Yaskawa INFORM job: GAUSSIANMOVING2.JBI

/JOB
//NAME GAUSSIANMOVING2
//POS
///NPOS 0,0,0,121,0,0
///TOOL 0
///POSTYPE ROBOT
///RECTAN
///RCONF 0,0,0,0,0,0,0,0,0,0,0,0,0,0,0,0,0,0,0,0,0,0,0,0
P00000=10.000,0.000,0.000,0.0000,0.0000,0.0000
///POSTYPE BASE
///TOOL0
P00001=0652.35187878,0006.95945011,0523.09500000,0000.00000000,0000.00400000,0180.00000000,
P00002=0652.29694326,0006.95464388,0523.09500000,0000.00000000,0000.00400000,0180.00000000,
P00003=0652.22427337,0006.94828609,0523.09500000,0000.00000000,0000.00400000,0180.00000000,
P00004=0652.12909978,0006.93995948,0523.09500000,0000.00000000,0000.00400000,0180.00000000,
P00005=0652.00569299,0006.92916278,0523.09500000,0000.00000000,0000.00400000,0180.00000000,
P00006=0651.84726850,0006.91530243,0523.09500000,0000.00000000,0000.00400000,0180.00000000,
P00007=0651.64591172,0006.89768600,0523.09500000,0000.00000000,0000.00400000,0180.00000000,
P00008=0651.39253259,0006.87551820,0523.09500000,0000.00000000,0000.00400000,0180.00000000,
P00009=0651.07686056,0006.84790047,0523.09500000,0000.00000000,0000.00400000,0180.00000000,
P00010=0650.68749098,0006.81383505,0523.09500000,0000.00000000,0000.00400000,0180.00000000,
P00011=0650.21199308,0006.77223437,0523.09500000,0000.00000000,0000.00400000,0180.00000000,
P00012=0649.63708838,0006.72193673,0523.09500000,0000.00000000,0000.00400000,0180.00000000,
P00013=0648.94890563,0006.66172854,0523.09500000,0000.00000000,0000.00400000,0180.00000000,
P00014=0648.13331474,0006.59037358,0523.09500000,0000.00000000,0000.00400000,0180.00000000,
P00015=0647.17633747,0006.50664892,0523.09500000,0000.00000000,0000.00400000,0180.00000000,
P00016=0646.06462739,0006.40938689,0523.09500000,0000.00000000,0000.00400000,0180.00000000,
P00017=0644.78600549,0006.29752197,0523.09500000,0000.00000000,0000.00400000,0180.00000000,
P00018=0643.33003222,0006.17014081,0523.09500000,0000.00000000,0000.00400000,0180.00000000,
P00019=0641.68859100,0006.02653332,0523.09500000,0000.00000000,0000.00400000,0180.00000000,
P00020=0639.85645402,0005.86624210,0523.09500000,0000.00000000,0000.00400000,0180.00000000,
P00021=0637.83179817,0005.68910767,0523.09500000,0000.00000000,0000.00400000,0180.00000000,
P00022=0635.61663786,0005.49530625,0523.09500000,0000.00000000,0000.00400000,0180.00000000,
P00023=0633.21714325,0005.28537767,0523.09500000,0000.00000000,0000.00400000,0180.00000000,
P00024=0630.64381570,0005.06024069,0523.09500000,0000.00000000,0000.00400000,0180.00000000,
P00025=0627.91149903,0004.82119395,0523.09500000,0000.00000000,0000.00400000,0180.00000000,
P00026=0625.03921312,0004.56990150,0523.09500000,0000.00000000,0000.00400000,0180.00000000,
P00027=0622.04980661,0004.30836232,0523.09500000,0000.00000000,0000.00400000,0180.00000000,
P00028=0618.96943611,0004.03886482,0523.09500000,0000.00000000,0000.00400000,0180.00000000,
P00029=0615.82689035,0003.76392769,0523.09500000,0000.00000000,0000.00400000,0180.00000000,
P00030=0612.65278792,0003.48622971,0523.09500000,0000.00000000,0000.00400000,0180.00000000,
P00031=0609.47868550,0003.20853173,0523.09500000,0000.00000000,0000.00400000,0180.00000000,
P00032=0606.33613974,0002.93359460,0523.09500000,0000.00000000,0000.00400000,0180.00000000,
P00033=0603.25576923,0002.66409710,0523.09500000,0000.00000000,0000.00400000,0180.00000000,
P00034=0600.26636273,0002.40255792,0523.09500000,0000.00000000,0000.00400000,0180.00000000,
P00035=0597.39407682,0002.15126547,0523.09500000,0000.00000000,0000.00400000,0180.00000000,
P00036=0594.66176015,0001.91221873,0523.09500000,0000.00000000,0000.00400000,0180.00000000,
P00037=0592.08843260,0001.68708175,0523.09500000,0000.00000000,0000.00400000,0180.00000000,
P00038=0589.68893799,0001.47715317,0523.09500000,0000.00000000,0000.00400000,0180.00000000,
P00039=0587.47377768,0001.28335175,0523.09500000,0000.00000000,0000.00400000,0180.00000000,
P00040=0585.44912182,0001.10621732,0523.09500000,0000.00000000,0000.00400000,0180.00000000,
P00041=0583.61698485,0000.94592610,0523.09500000,0000.00000000,0000.00400000,0180.00000000,
P00042=0581.97554363,0000.80231861,0523.09500000,0000.00000000,0000.00400000,0180.00000000,
P00043=0580.51957036,0000.67493745,0523.09500000,0000.00000000,0000.00400000,0180.00000000,
P00044=0579.24094846,0000.56307253,0523.09500000,0000.00000000,0000.00400000,0180.00000000,
P00045=0578.12923838,0000.46581050,0523.09500000,0000.00000000,0000.00400000,0180.00000000,
P00046=0577.17226111,0000.38208584,0523.09500000,0000.00000000,0000.00400000,0180.00000000,
P00047=0576.35667022,0000.31073088,0523.09500000,0000.00000000,0000.00400000,0180.00000000,
P00048=0575.66848747,0000.25052269,0523.09500000,0000.00000000,0000.00400000,0180.00000000,
P00049=0575.09358277,0000.20022505,0523.09500000,0000.00000000,0000.00400000,0180.00000000,
P00050=0574.61808487,0000.15862437,0523.09500000,0000.00000000,0000.00400000,0180.00000000,
P00051=0574.22871528,0000.12455895,0523.09500000,0000.00000000,0000.00400000,0180.00000000,
P00052=0573.91304326,0000.09694122,0523.09500000,0000.00000000,0000.00400000,0180.00000000,
P00053=0573.65966412,0000.07477342,0523.09500000,0000.00000000,0000.00400000,0180.00000000,
P00054=0573.45830735,0000.05715699,0523.09500000,0000.00000000,0000.00400000,0180.00000000,
P00055=0573.29988285,0000.04329664,0523.09500000,0000.00000000,0000.00400000,0180.00000000,
P00056=0573.17647606,0000.03249994,0523.09500000,0000.00000000,0000.00400000,0180.00000000,
P00057=0573.08130247,0000.02417333,0523.09500000,0000.00000000,0000.00400000,0180.00000000,
P00058=0573.00863258,0000.01781554,0523.09500000,0000.00000000,0000.00400000,0180.00000000,
P00059=0572.95369707,0000.01300931,0523.09500000,0000.00000000,0000.00400000,0180.00000000,
P00060=0572.91258090,0000.00941211,0523.09500000,0000.00000000,0000.00400000,0180.00000000,
///TOOL1
P00061=0667.35246409,0026.78692869,0908.48000000,0180.00000000,0000.00000000,0000.00000000
P00062=0667.35742094,0026.76842948,0908.48000000,0180.00000000,0000.00000000,0000.00000000
P00063=0667.36397796,0026.74395834,0908.48000000,0180.00000000,0000.00000000,0000.00000000
P00064=0667.37256550,0026.71190921,0908.48000000,0180.00000000,0000.00000000,0000.00000000
P00065=0667.38370053,0026.67035272,0908.48000000,0180.00000000,0000.00000000,0000.00000000
P00066=0667.39799521,0026.61700424,0908.48000000,0180.00000000,0000.00000000,0000.00000000
P00067=0667.41616369,0026.54919856,0908.48000000,0180.00000000,0000.00000000,0000.00000000
P00068=0667.43902615,0026.46387468,0908.48000000,0180.00000000,0000.00000000,0000.00000000
P00069=0667.46750932,0026.35757404,0908.48000000,0180.00000000,0000.00000000,0000.00000000
P00070=0667.50264224,0026.22645619,0908.48000000,0180.00000000,0000.00000000,0000.00000000
P00071=0667.54554654,0026.06633516,0908.48000000,0180.00000000,0000.00000000,0000.00000000
P00072=0667.59742035,0025.87273949,0908.48000000,0180.00000000,0000.00000000,0000.00000000
P00073=0667.65951526,0025.64099813,0908.48000000,0180.00000000,0000.00000000,0000.00000000
P00074=0667.73310624,0025.36635284,0908.48000000,0180.00000000,0000.00000000,0000.00000000
P00075=0667.81945455,0025.04409656,0908.48000000,0180.00000000,0000.00000000,0000.00000000
P00076=0667.91976445,0024.66973493,0908.48000000,0180.00000000,0000.00000000,0000.00000000
P00077=0668.03513484,0024.23916677,0908.48000000,0180.00000000,0000.00000000,0000.00000000
P00078=0668.16650769,0023.74887660,0908.48000000,0180.00000000,0000.00000000,0000.00000000
P00079=0668.31461537,0023.19613124,0908.48000000,0180.00000000,0000.00000000,0000.00000000
P00080=0668.47992957,0022.57917023,0908.48000000,0180.00000000,0000.00000000,0000.00000000
P00081=0668.66261480,0021.89737966,0908.48000000,0180.00000000,0000.00000000,0000.00000000
P00082=0668.86248931,0021.15143787,0908.48000000,0180.00000000,0000.00000000,0000.00000000
P00083=0669.07899634,0020.34342262,0908.48000000,0180.00000000,0000.00000000,0000.00000000
P00084=0669.31118836,0019.47687018,0908.48000000,0180.00000000,0000.00000000,0000.00000000
P00085=0669.55772602,0018.55677912,0908.48000000,0180.00000000,0000.00000000,0000.00000000
P00086=0669.81689314,0017.58955428,0908.48000000,0180.00000000,0000.00000000,0000.00000000
P00087=0670.08662808,0016.58288978,0908.48000000,0180.00000000,0000.00000000,0000.00000000
P00088=0670.36457072,0015.54559370,0908.48000000,0180.00000000,0000.00000000,0000.00000000
P00089=0670.64812346,0014.48736049,0908.48000000,0180.00000000,0000.00000000,0000.00000000
P00090=0670.93452356,0013.41850076,0908.48000000,0180.00000000,0000.00000000,0000.00000000
P00091=0671.22092366,0012.34964103,0908.48000000,0180.00000000,0000.00000000,0000.00000000
P00092=0671.50447639,0011.29140782,0908.48000000,0180.00000000,0000.00000000,0000.00000000
P00093=0671.78241904,0010.25411174,0908.48000000,0180.00000000,0000.00000000,0000.00000000
P00094=0672.05215398,0009.24744724,0908.48000000,0180.00000000,0000.00000000,0000.00000000
P00095=0672.31132110,0008.28022240,0908.48000000,0180.00000000,0000.00000000,0000.00000000
P00096=0672.55785875,0007.36013134,0908.48000000,0180.00000000,0000.00000000,0000.00000000
P00097=0672.79005078,0006.49357890,0908.48000000,0180.00000000,0000.00000000,0000.00000000
P00098=0673.00655781,0005.68556365,0908.48000000,0180.00000000,0000.00000000,0000.00000000
P00099=0673.20643231,0004.93962186,0908.48000000,0180.00000000,0000.00000000,0000.00000000
P00100=0673.38911754,0004.25783129,0908.48000000,0180.00000000,0000.00000000,0000.00000000
P00101=0673.55443175,0003.64087028,0908.48000000,0180.00000000,0000.00000000,0000.00000000
P00102=0673.70253942,0003.08812491,0908.48000000,0180.00000000,0000.00000000,0000.00000000
P00103=0673.83391228,0002.59783475,0908.48000000,0180.00000000,0000.00000000,0000.00000000
P00104=0673.94928267,0002.16726659,0908.48000000,0180.00000000,0000.00000000,0000.00000000
P00105=0674.04959256,0001.79290496,0908.48000000,0180.00000000,0000.00000000,0000.00000000
P00106=0674.13594088,0001.47064867,0908.48000000,0180.00000000,0000.00000000,0000.00000000
P00107=0674.20953186,0001.19600339,0908.48000000,0180.00000000,0000.00000000,0000.00000000
P00108=0674.27162677,0000.96426203,0908.48000000,0180.00000000,0000.00000000,0000.00000000
P00109=0674.32350057,0000.77066636,0908.48000000,0180.00000000,0000.00000000,0000.00000000
P00110=0674.36640487,0000.61054533,0908.48000000,0180.00000000,0000.00000000,0000.00000000
P00111=0674.40153779,0000.47942748,0908.48000000,0180.00000000,0000.00000000,0000.00000000
P00112=0674.43002096,0000.37312684,0908.48000000,0180.00000000,0000.00000000,0000.00000000
P00113=0674.45288343,0000.28780296,0908.48000000,0180.00000000,0000.00000000,0000.00000000
P00114=0674.47105191,0000.21999728,0908.48000000,0180.00000000,0000.00000000,0000.00000000
P00115=0674.48534659,0000.16664880,0908.48000000,0180.00000000,0000.00000000,0000.00000000
P00116=0674.49648162,0000.12509231,0908.48000000,0180.00000000,0000.00000000,0000.00000000
P00117=0674.50506915,0000.09304318,0908.48000000,0180.00000000,0000.00000000,0000.00000000
P00118=0674.51162618,0000.06857204,0908.48000000,0180.00000000,0000.00000000,0000.00000000
P00119=0674.51658302,0000.05007283,0908.48000000,0180.00000000,0000.00000000,0000.00000000
P00120=0674.52029295,0000.03622722,0908.48000000,0180.00000000,0000.00000000,0000.00000000
//INST
///DATE 2017/03/31 08:11
///COMM PLAYINGTWOROBOTS
///ATTR SC,RW
///GROUP1 RB1
///GROUP2 RB2
NOP
DOUT OT#(16) OFF
DOUT OT#(15) ON
DOUT OT#(16) ON
MOVL P00001 V=0003.4465852  +MOVL P00061 V=0001.1969865
MOVL P00002 V=0004.5592174  +MOVL P00062 V=0001.5833996
MOVL P00003 V=0005.9710711  +MOVL P00063 V=0002.0737312
MOVL P00004 V=0007.7423865  +MOVL P00064 V=0002.6889026
MOVL P00005 V=0009.9393530  +MOVL P00065 V=0003.4519011
MOVL P00006 V=0012.6328705  +MOVL P00066 V=0004.3873499
MOVL P00007 V=0015.8966875  +MOVL P00067 V=0005.5208616
MOVL P00008 V=0019.8048652  +MOVL P00068 V=0006.8781575
MOVL P00009 V=0024.4285569  +MOVL P00069 V=0008.4839488
MOVL P00010 V=0029.8321393  +MOVL P00070 V=0010.3605933
MOVL P00011 V=0036.0687965  +MOVL P00071 V=0012.5265616
MOVL P00012 V=0043.1757182  +MOVL P00072 V=0014.9947696
MOVL P00013 V=0051.1691447  +MOVL P00073 V=0017.7708575
MOVL P00014 V=0060.0395478  +MOVL P00074 V=0020.8515161
MOVL P00015 V=0069.7472898  +MOVL P00075 V=0024.2229796
MOVL P00016 V=0080.2191268  +MOVL P00076 V=0027.8598104
MOVL P00017 V=0091.3459282  +MOVL P00077 V=0031.7241079
MOVL P00018 V=0102.9819536  +MOVL P00078 V=0035.7652572
MOVL P00019 V=0114.9459649  +MOVL P00079 V=0039.9203147
MOVL P00020 V=0127.0243571  +MOVL P00080 V=0044.1150963
MOVL P00021 V=0138.9763662  +MOVL P00081 V=0048.2659855
MOVL P00022 V=0150.5412682  +MOVL P00082 V=0052.2824338
MOVL P00023 V=0161.4473276  +MOVL P00083 V=0056.0700685
MOVL P00024 V=0171.4221049  +MOVL P00084 V=0059.5342722
MOVL P00025 V=0180.2035983  +MOVL P00085 V=0062.5840529
MOVL P00026 V=0187.5515971  +MOVL P00086 V=0065.1359861
MOVL P00027 V=0193.2585637  +MOVL P00087 V=0067.1179948
MOVL P00028 V=0197.1593608  +MOVL P00088 V=0068.4727274
MOVL P00029 V=0199.1391864  +MOVL P00089 V=0069.1603136
MOVL P00030 V=0199.1391864  +MOVL P00090 V=0069.1603136
MOVL P00031 V=0197.1593608  +MOVL P00091 V=0068.4727274
MOVL P00032 V=0193.2585637  +MOVL P00092 V=0067.1179948
MOVL P00033 V=0187.5515971  +MOVL P00093 V=0065.1359861
MOVL P00034 V=0180.2035983  +MOVL P00094 V=0062.5840529
MOVL P00035 V=0171.4221049  +MOVL P00095 V=0059.5342722
MOVL P00036 V=0161.4473276  +MOVL P00096 V=0056.0700685
MOVL P00037 V=0150.5412682  +MOVL P00097 V=0052.2824338
MOVL P00038 V=0138.9763662  +MOVL P00098 V=0048.2659855
MOVL P00039 V=0127.0243571  +MOVL P00099 V=0044.1150963
MOVL P00040 V=0114.9459649  +MOVL P00100 V=0039.9203147
MOVL P00041 V=0102.9819536  +MOVL P00101 V=0035.7652572
MOVL P00042 V=0091.3459282  +MOVL P00102 V=0031.7241079
MOVL P00043 V=0080.2191268  +MOVL P00103 V=0027.8598104
MOVL P00044 V=0069.7472898  +MOVL P00104 V=0024.2229796
MOVL P00045 V=0060.0395478  +MOVL P00105 V=0020.8515161
MOVL P00046 V=0051.1691447  +MOVL P00106 V=0017.7708575
MOVL P00047 V=0043.1757182  +MOVL P00107 V=0014.9947696
MOVL P00048 V=0036.0687965  +MOVL P00108 V=0012.5265616
MOVL P00049 V=0029.8321393  +MOVL P00109 V=0010.3605933
MOVL P00050 V=0024.4285569  +MOVL P00110 V=0008.4839488
MOVL P00051 V=0019.8048652  +MOVL P00111 V=0006.8781575
MOVL P00052 V=0015.8966875  +MOVL P00112 V=0005.5208616
MOVL P00053 V=0012.6328705  +MOVL P00113 V=0004.3873499
MOVL P00054 V=0009.9393530  +MOVL P00114 V=0003.4519011
MOVL P00055 V=0007.7423865  +MOVL P00115 V=0002.6889026
MOVL P00056 V=0005.9710711  +MOVL P00116 V=0002.0737312
MOVL P00057 V=0004.5592174  +MOVL P00117 V=0001.5833996
MOVL P00058 V=0003.4465852  +MOVL P00118 V=0001.1969865
MOVL P00059 V=0002.5795763  +MOVL P00119 V=0000.8958775
MOVL P00060 V=0002.5795763  +MOVL P00120 V=0000.8958775
DOUT OT#(16) OFF
DOUT OT#(15) OFF
DOUT OT#(16) ON
END
